// TIA Portal V20 export
TYPE "typeSequenceControlNode"
// stored: Namespace Unit1.Em13
   STRUCT
      jobs : "LAF_typeJobs";
      sequence : "LAF_typeSequence";
      selectJobStatus { S7_SetPoint := 'True'} : Array[0..10] of "LAF_typeJobStatus";
      "step" : "LER_typeStep";
      jobInterface : "Unit1.Em13.typeSequenceControlNodeJobInterface";
      homeCheck : "Unit1.Em13.typeSequenceControlNodeHomeCheck";
   END_STRUCT;
   // // "step".action1[101] : Step[101] : JOB[1] Condition
   // // "step".action1[110] : Step[110] : Clamp Open
   // // "step".action1[150] : Step[150] : JR Unload P&P X-axis Work Ready Position
   // // "step".action1[160] : Step[160] : JR Unload P&P Z-axis Wait Position
   // // "step".action1[170] : Step[170] : JR Unload P&P X-axis Wait Position
   // // "step".action1[180] : Step[180] : JR Unload P&P C-axis Wait Position
   // // "step".action1[190] : Step[190] : JOB[1] Step End
   // // "step".action1[201] : Step[201] : JOB[2] Condition
   // // "step".action1[210] : Step[210] : JR Unload P&P C-axis Weight Check Position
   // // "step".action1[220] : Step[220] : JR Unload P&P X-axis Work Ready Position
   // // "step".action1[230] : Step[230] : JR Unload P&P Z-axis Weight Check Position
   // // "step".action1[240] : Step[240] : JR Unload P&P X-axis Weight Check Position
   // // "step".action1[250] : Step[250] : Clamp Close
   // // "step".action1[290] : Step[290] : JOB[2] Step End
   // // "step".action1[301] : Step[301] : JOB[3] Condition
   // // "step".action1[310] : Step[310] : JR Unload P&P X-axis Work Ready Position
   // // "step".action1[320] : Step[320] : JR Unload P&P Z-axis Wait Position
   // // "step".action1[330] : Step[330] : JR Unload P&P X-axis Wait Position
   // // "step".action1[340] : Step[340] : JR Unload P&P C-axis Packaging Position
   // // "step".action1[350] : Step[350] : JR Unload P&P Z-axis Packaging Position
   // // "step".action1[360] : Step[360] : JR Unload P&P X-axis Packaging Position
   // // "step".action1[370] : Step[370] : Clamp Open
   // // "step".action1[380] : Step[380] : JR Unload P&P X/Z/C-Axis Wait Position
   // // "step".action1[390] : Step[390] : Job3 Step End
   // // "step".action1[401] : Step[401] : JOB[4] Condition
   // // "step".action1[410] : Step[410] : JR Unload P&P C-axis Stack NG Box Position
   // // "step".action1[411] : STEP[411] : JR Unload P&P X-axis Work Ready Position
   // // "step".action1[420] : STEP[420] : JR Unload P&P Z-axis Stack NG Box Position
   // // "step".action1[430] : STEP[430] : JR Unload P&P X-axis Stack NG Box Position
   // // "step".action1[431] : STEP[431] : JR Unloading P&P [Unloading Ready] => Stack NG Box
   // // "step".action1[440] : STEP[440] : Clamp Open
   // // "step".action1[450] : STEP[450] : JR Unload P&P X-axis Work Ready Position
   // // "step".action1[480] : STEP[480] : JR Unload P&P X/Z/C-Axis Wait Position
   // // "step".action1[490] : STEP[490] : JOB[4] Step End
   // // "step".transition1[101] : Step[101] : JOB[1] Condition
   // // "step".transition1[110] : Step[110] : Clamp Open
   // // "step".transition1[150] : Step[150] : JR Unload P&P X-axis Work Ready Position
   // // "step".transition1[160] : Step[160] : JR Unload P&P Z-axis Wait Position
   // // "step".transition1[170] : Step[170] : JR Unload P&P X-axis Wait Position
   // // "step".transition1[180] : Step[180] : JR Unload P&P C-axis Wait Position
   // // "step".transition1[190] : Step[190] : JOB[1] Step End
   // // "step".transition1[201] : Step[201] : JOB[2] Condition
   // // "step".transition1[210] : Step[210] : JR Unload P&P C-axis Weight Check Position
   // // "step".transition1[220] : Step[220] : JR Unload P&P X-axis Work Ready Position
   // // "step".transition1[230] : Step[230] : JR Unload P&P Z-axis Weight Check Position
   // // "step".transition1[240] : Step[240] : JR Unload P&P X-axis Weight Check Position
   // // "step".transition1[250] : Step[250] : Clamp Close
   // // "step".transition1[290] : Step[290] : JOB[2] Step End
   // // "step".transition1[301] : Step[301] : JOB[3] Condition
   // // "step".transition1[310] : Step[310] : JR Unload P&P X-axis Work Ready Position
   // // "step".transition1[320] : Step[320] : JR Unload P&P Z-axis Wait Position
   // // "step".transition1[330] : Step[330] : JR Unload P&P X-axis Wait Position
   // // "step".transition1[340] : Step[340] : JR Unload P&P C-axis Packaging Position
   // // "step".transition1[350] : Step[350] : JR Unload P&P Z-axis Packaging Position
   // // "step".transition1[360] : Step[360] : JR Unload P&P X-axis Packaging Position
   // // "step".transition1[370] : Step[370] : Clamp Open
   // // "step".transition1[380] : Step[380] : JR Unload P&P X/Z/C-Axis Wait Position
   // // "step".transition1[390] : Step[390] : Job3 Step End
   // // "step".transition1[401] : Step[401] : JOB[4] Condition
   // // "step".transition1[410] : Step[410] : JR Unload P&P C-axis Stack NG Box Position
   // // "step".transition1[411] : STEP[411] : JR Unload P&P X-axis Work Ready Position
   // // "step".transition1[420] : STEP[420] : JR Unload P&P Z-axis Stack NG Box Position
   // // "step".transition1[430] : STEP[430] : JR Unload P&P X-axis Stack NG Box Position
   // // "step".transition1[431] : STEP[431] : JR Unloading P&P [Unloading Ready] => Stack NG Box
   // // "step".transition1[440] : STEP[440] : Clamp Open
   // // "step".transition1[450] : STEP[450] : JR Unload P&P X-axis Work Ready Position
   // // "step".transition1[480] : STEP[480] : JR Unload P&P X/Z/C-Axis Wait Position
   // // "step".transition1[490] : STEP[490] : JOB[4] Step End
END_TYPE
